(* CoDeSys 2.3 export: POWEREDBYGENERATOR.EXP *)

(* POU Steuerung/PoweredByGenerator, ST *)
PROGRAM PoweredByGenerator
VAR_INPUT
	init: BOOL;
END_VAR
VAR
	rtTaste: R_TRIG;
	tofTaste: TOF;
END_VAR
IF init THEN
	(* Nach dem Einschalten erst mal aktivieren *)
	outputs.SchuetzGrundlast := TRUE;
END_IF

(* Taste entprellen *)
tofTaste(IN := inputs.TastePoweredByGenerator, PT := T#200ms);
rtTaste(CLK := tofTaste.Q);
IF rtTaste.Q THEN
	(* toggle *)
	outputs.SchuetzGrundlast := NOT outputs.SchuetzGrundlast;
END_IF
END_PROGRAM
